Staubli VAL3: Joint2Point.pgx

public program Joint2Point(jointRx x_jJSource, pointRx& x_pP)
begin
  //把joint点转换为point
  //movel与movej之间相互转换

  x_pP=jointToPoint(TxtFile:tCfg,world,x_jJSource)
  //x_pP.trsf=x_pP.trsf*!TxtFile:fProduct.trsf*!TxtFile:fTraj.trsf
  x_pP.trsf=!TxtFile:fTraj.trsf*!TxtFile:fProduct.trsf*x_pP.trsf
  link(x_pP,TxtFile:fArray)








end
